FUNCTION_BLOCK CAerationLogicBasic (* Basic Function Block Type *)
  (* Standard: 61499-2 *)
  (* Version 1.0, 9/29/2026, Schneider Electric, Rev1 - ECC executa tambem em VALVEBLOWER_RDY (valvula do B1/B4 voltando ao automatico) *)
  PACKAGE SE.Nereda;
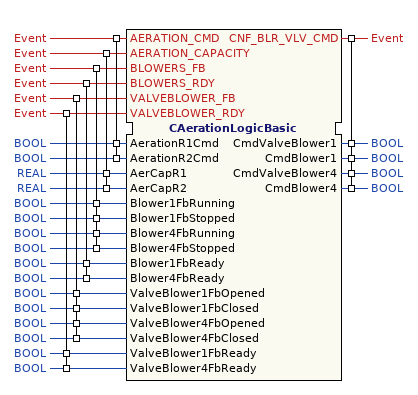
  EVENT_INPUT
    AERATION_CMD WITH AerationR1Cmd, AerationR2Cmd;
    AERATION_CAPACITY WITH AerCapR1, AerCapR2;
    BLOWERS_FB WITH Blower1FbRunning, Blower1FbStopped, Blower4FbRunning, Blower4FbStopped;
    BLOWERS_RDY WITH Blower1FbReady, Blower4FbReady;
    VALVEBLOWER_FB WITH ValveBlower1FbOpened, ValveBlower1FbClosed, ValveBlower4FbOpened, ValveBlower4FbClosed;
    VALVEBLOWER_RDY WITH ValveBlower1FbReady, ValveBlower4FbReady;
  END_EVENT
  EVENT_OUTPUT
    CNF_BLR_VLV_CMD WITH CmdBlower1, CmdBlower4, CmdValveBlower1, CmdValveBlower4;
  END_EVENT
  VAR_INPUT
    AerationR1Cmd : BOOL;
    AerationR2Cmd : BOOL;
    AerCapR1 : REAL;
    AerCapR2 : REAL;
    Blower1FbRunning : BOOL;
    Blower1FbStopped : BOOL;
    Blower4FbRunning : BOOL;
    Blower4FbStopped : BOOL;
    Blower1FbReady : BOOL;
    Blower4FbReady : BOOL;
    ValveBlower1FbOpened : BOOL;
    ValveBlower1FbClosed : BOOL;
    ValveBlower4FbOpened : BOOL;
    ValveBlower4FbClosed : BOOL;
    ValveBlower1FbReady : BOOL;
    ValveBlower4FbReady : BOOL;
  END_VAR
  VAR_OUTPUT
    CmdValveBlower1 : BOOL;
    CmdBlower1 : BOOL;
    CmdValveBlower4 : BOOL;
    CmdBlower4 : BOOL;
  END_VAR
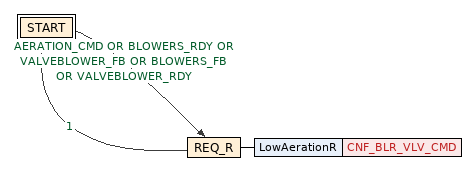
  EC_STATES
    START; (* Initial State *)
    REQ_R : LowAerationR -> CNF_BLR_VLV_CMD;
  END_STATES
  EC_TRANSITIONS
    START TO REQ_R := AERATION_CMD OR BLOWERS_RDY OR VALVEBLOWER_FB OR BLOWERS_FB OR VALVEBLOWER_RDY;
    REQ_R TO START := 1;
  END_TRANSITIONS
  ALGORITHM LowAerationR IN ST:
;
IF AerationR1Cmd AND ValveBlower1FbReady THEN
	CmdValveBlower1 := TRUE;
ELSIF Blower1FbStopped THEN
	CmdValveBlower1 := FALSE;
END_IF;

IF AerationR2Cmd AND ValveBlower4FbReady THEN
	CmdValveBlower4 := TRUE;
ELSIF Blower4FbStopped THEN
	CmdValveBlower4 := FALSE;
END_IF;

IF AerationR1Cmd AND Blower1FbReady AND ValveBlower1FbOpened THEN
	CmdBlower1 := TRUE;
ELSE
	CmdBlower1 := FALSE;
END_IF;

IF AerationR2Cmd AND Blower4FbReady AND ValveBlower4FbOpened THEN
	CmdBlower4 := TRUE;
ELSE
	CmdBlower4 := FALSE;
END_IF;

IF Blower4FbStopped AND NOT Blower4FbReady THEN
	CmdValveBlower4 := FALSE;
END_IF;

IF Blower1FbStopped AND NOT Blower1FbReady THEN
	CmdValveBlower1 := FALSE;
END_IF;
  END_ALGORITHM
  ALGORITHM OpenValve IN ST:
;

IF AerationR1Cmd AND ValveBlower1FbReady THEN
	CmdValveBlower1 := TRUE;
ELSE
	CmdValveBlower1 := FALSE;
END_IF;

IF AerationR2Cmd AND ValveBlower4FbReady THEN
	CmdValveBlower4 := TRUE;
ELSE
	CmdValveBlower4 := FALSE;
END_IF;

IF AerationR1Cmd AND Blower1FbReady AND ValveBlower1FbOpened THEN
	CmdBlower1 := TRUE;
ELSE
	CmdBlower1 := FALSE;
END_IF;

IF AerationR2Cmd AND Blower4FbReady AND ValveBlower4FbOpened THEN
	CmdBlower4 := TRUE;
ELSE
	CmdBlower4 := FALSE;
END_IF;
  END_ALGORITHM
END_FUNCTION_BLOCK
